// TIA Portal project "Paketband_6" (V20)

(* hardware
DEVICE "S7-1500/ET200MP-Station_1"  S7-1500 station
   slot 0: "Profilschiene_0"  Rack  6ES7 590-1***0-0AA0
   slot 1: "PLC_1"  CPU 1513-1 PN  6ES7 513-1AM03-0AB0  V4.0
      slot 3: "CPU-Display_1"  6ES7591-1AA00-0AA0
      slot 32768: "PROFINET-Schnittstelle_1"  X1
         slot 32769: "Port_1"  X1 P1
         slot 32770: "Port_2"  X1 P2
      slot 34817: "Virtual CP interface port_1"  Virtual CP interface port  Virtual CP interface port FW V4.0
   slot 2: "DI 16x24VDC BA_1"  DI 16x24VDC BA  6ES7 521-1BH10-0AA0  V1.1
   slot 3: "DQ 16x24VDC/0.5A ST_1"  DQ 16x24VDC/0.5A ST  6ES7 522-1BH00-0AB0  V2.0
   slot 4: "AI 8xU/I/R/RTD BA_1"  AI 8xU/I/R/RTD BA  6ES7 531-7QF00-0AB0  V1.0
   slot 5: "AQ 8xU/I HS_1"  AQ 8xU/I HS  6ES7 532-5HF00-0AB0  V2.2
   slot 6: "AQ 2xU/I ST_1"  AQ 2xU/I ST  6ES7 532-5NB00-0AB0  V1.0
*)

// ===== PLC "PLC_1"  CPU 1513-1 PN =====

VAR_GLOBAL   // PLC tag table "Standard-Variablentabelle"
   "PlcLabConnectIn01" AT %ID32760 : DWord;
   "PlcLabConnectIn02" AT %ID32764 : DWord;
   "PlcLabConnectOut01" AT %QD32760 : DWord;
   "PlcLabConnectOut02" AT %QD32764 : DWord;
   "Förderband_an" AT %M1.2 : Bool;
   "Förderband_aus" AT %M1.3 : Bool;
   "NotAus_aktiv" AT %M1.1 : Bool;
   "Anlage_ein" AT %M1.0 : Bool;
   "Paket_erkannt" AT %M1.4 : Bool;
   "Temp_1" AT %M0.0 : Bool;
   "Temp_2" AT %M0.1 : Bool;
   "Clock_Byte" AT %MB100 : Byte;
   "Clock_10Hz" AT %M100.0 : Bool;
   "Clock_5Hz" AT %M100.1 : Bool;
   "Clock_2.5Hz" AT %M100.2 : Bool;
   "Clock_2Hz" AT %M100.3 : Bool;
   "Clock_1.25Hz" AT %M100.4 : Bool;
   "Clock_1Hz" AT %M100.5 : Bool;
   "Clock_0.625Hz" AT %M100.6 : Bool;
   "Clock_0.5Hz" AT %M100.7 : Bool;
   "Förderband_starten" AT %M1.5 : Bool;
   "Paketzahl_erreicht" AT %M1.6 : Bool;
END_VAR

VAR_GLOBAL   // PLC tag table "Eingänge"
   "S1" AT %E0.4 : Bool;   // Start-Taster
   "S2" AT %E0.5 : Bool;   // Stopp-Taster
   "S4" AT %E0.0 : Bool;   // Not-Aus Schalter
   "S0" AT %E0.1 : Bool;   // Betriebsschalter auf ein
   "S3" AT %E0.6 : Bool;   // Rücksetz-Taster
   "S5" AT %E1.0 : Bool;   // Wiedereinschalten Taster
   "1b1" AT %E1.1 : Bool;   // Lichttaster (Mitte)
   "2b1" AT %E1.2 : Bool;   // Lichttaster (Ende)
   "S6" AT %E0.7 : Bool;   // Wartung quittieren Taster
END_VAR

VAR_GLOBAL   // PLC tag table "Ausgänge"
   "S1_Licht" AT %A0.4 : Bool;   // Lampe des Start-Tasters
   "S2_Licht" AT %A0.5 : Bool;   // Lampe des Stopp-Tasters
   "M1" AT %A0.0 : Bool;   // Förderband
   "S3_Licht" AT %A0.6 : Bool;   // Lampe des Rücksetz-Tasters
   "H1" AT %A0.1 : Bool;   // Meldeleuchte (Grün)
   "H2" AT %A0.2 : Bool;   // Meldeleuchte (Gelb)
   "H3" AT %A0.3 : Bool;   // Meldeleuchte (Rot)
   "Rundumleuchte" AT %A0.7 : Bool;
   "Zähler" AT %AW30 : Int;
   "H4" AT %A1.0 : Bool;   // Meldeleuchte (Blau)
END_VAR

// folder: System blocks/Program resources

DATA_BLOCK "DB_Timer_EV_3s"   // DB1
{ S7_Optimized_Access := 'TRUE' }
AUTHOR : Simatic
FAMILY : IEC
NAME : IEC_TMR
VERSION : 1.0
// stored: InstanceOfName IEC_TIMER
"IEC_TIMER"
BEGIN
END_DATA_BLOCK

DATA_BLOCK "DB_Timer_10d_Wartung"   // DB2
{ S7_Optimized_Access := 'TRUE' }
AUTHOR : Simatic
FAMILY : IEC
NAME : IEC_TMR
VERSION : 1.0
// stored: InstanceOfName IEC_TIMER
"IEC_TIMER"
BEGIN
END_DATA_BLOCK

DATA_BLOCK "DB_Timer_EV_2s"   // DB3
{ S7_Optimized_Access := 'TRUE' }
AUTHOR : Simatic
FAMILY : IEC
NAME : IEC_TMR
VERSION : 1.0
// stored: InstanceOfName IEC_TIMER
"IEC_TIMER"
BEGIN
END_DATA_BLOCK

DATA_BLOCK "DB_Counter_Pakete"   // DB4
{ S7_Optimized_Access := 'TRUE' }
AUTHOR : Simatic
FAMILY : IEC
NAME : CNTR
VERSION : 1.0
// stored: InstanceOfName IEC_COUNTER
"IEC_COUNTER"
BEGIN
END_DATA_BLOCK

// folder: (top level)

FUNCTION "Paketbandanlage" : Void   // FC1, FBD
{ S7_Optimized_Access := 'FALSE' }
VERSION : 0.1
   VAR_TEMP   // added for the SCL form of the ladder/FBD networks
      _w1 : Bool;
      _w2 : Bool;
   END_VAR
BEGIN

REGION Network 1: Paketbandsteuerung
   // Hinweis: Alle Schalter können nur benutzt werden, wenn die Anlage über den Betriebsschalter eingeschaltet wurde.
   // Über S2 (Stopp-Taster), 1b1 bzw. 2b1 (Lichttaster) wird das Paketband gestoppt. Der Stopp-Modus, wird durch start des Förderbandes deaktiviert.
   // Beide Modi (Start, Stopp) werden deaktiviert, sobald S4 (Not-Aus Schalter) aktiv ist.
   // Der Not-Aus-Modus kann nur über S3 (Rücksetz-Taster) deaktiviert werden.
   // Nach 10 Tagen Laufzeit des Förderbandes soll das Band kontrolliert werden, dazu soll die Rundumleuchte dann angehen. Mit S6 (Rücksetztaster) soll die Wartung quittiert werden.
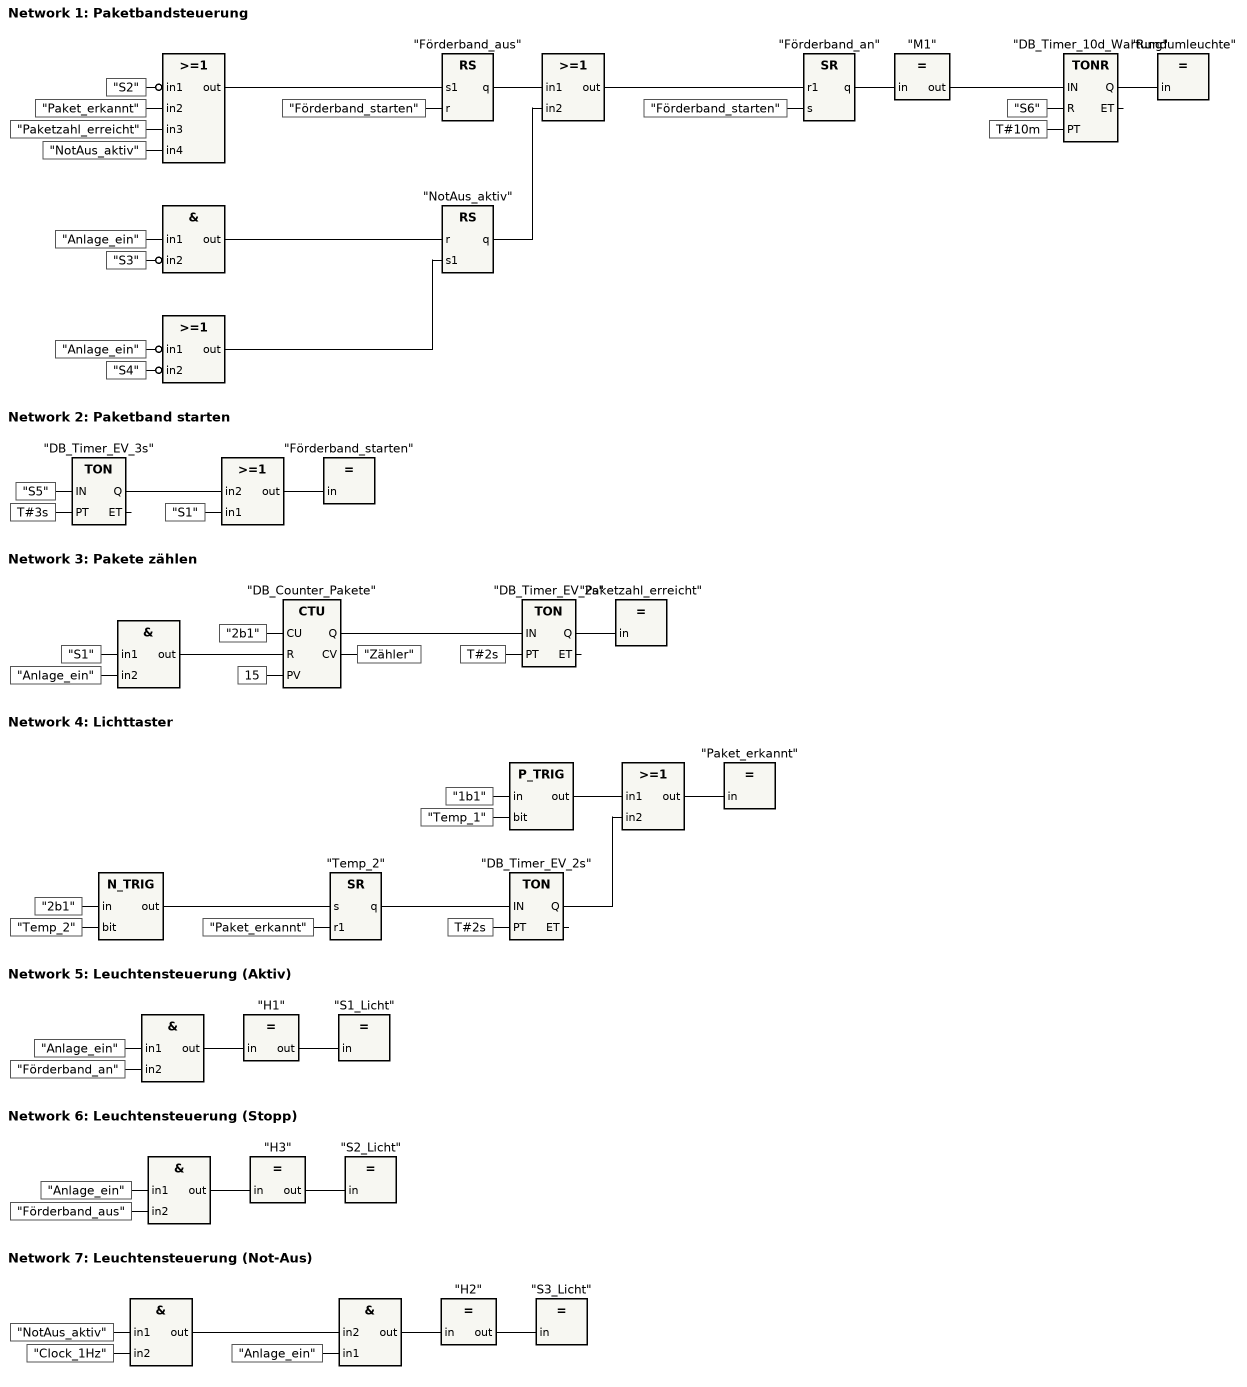
   IF "Förderband_starten" THEN
       "Förderband_aus" := FALSE;   // RS flip-flop
   END_IF;
   IF NOT "S2" OR "Paket_erkannt" OR "Paketzahl_erreicht" OR "NotAus_aktiv" THEN
       "Förderband_aus" := TRUE;
   END_IF;
   IF "Anlage_ein" AND NOT "S3" THEN
       "NotAus_aktiv" := FALSE;   // RS flip-flop
   END_IF;
   IF NOT "Anlage_ein" OR NOT "S4" THEN "NotAus_aktiv" := TRUE; END_IF;
   IF "Förderband_starten" THEN
       "Förderband_an" := TRUE;   // SR flip-flop
   END_IF;
   IF "Förderband_aus" OR "NotAus_aktiv" THEN "Förderband_an" := FALSE; END_IF;
   "M1" := "Förderband_an";
   "DB_Timer_10d_Wartung".TONR(IN := "Förderband_an", R := "S6", PT := T#10m);
   "Rundumleuchte" := "DB_Timer_10d_Wartung".Q;
END_REGION

REGION Network 2: Paketband starten
   // Das Paketband kann über S1 (Start-Taster) eingeschaltet werden bzw. durch S5 (Wiedereinschalten) und läuft dann dauerhaft. Der Schalter S5 (Wiedereinschalten) muss 3S gedrückt werden, bevor die Anlage wieder anlaufen darf. S1 (Starttaster) soll ganz normal funktionieren.
   "DB_Timer_EV_3s".TON(IN := "S5", PT := T#3s);
   "Förderband_starten" := "DB_Timer_EV_3s".Q OR "S1";
END_REGION

REGION Network 3: Pakete zählen
   // Nachdem 15 Pakete den hinteren Sensor durchlaufen haben, soll die Anlage automatisch abschalten. Über S1 (den Starttaster) soll der Zähler zurückgesetzt werden.
   "DB_Counter_Pakete".CTU(CU := "2b1", R := "S1" AND "Anlage_ein", PV := 15, CV => "Zähler");
   "DB_Timer_EV_2s".TON(IN := "DB_Counter_Pakete".Q, PT := T#2s);
   "Paketzahl_erreicht" := "DB_Timer_EV_2s".Q;
END_REGION

REGION Network 4: Lichttaster
   // Wenn 2b1 (der Lichttaster am Ende) oder 1b1 (Lichttaster in der Mitte) ein Paket erkennen, soll sofort bzw. verzögert das Band stehen bleiben.
   #_w1 := "1b1" AND NOT "Temp_1";   // rising edge
   "Temp_1" := "1b1";
   #_w2 := NOT "2b1" AND "Temp_2";   // falling edge
   "Temp_2" := "2b1";
   IF #_w2 THEN
       "Temp_2" := TRUE;   // SR flip-flop
   END_IF;
   IF "Paket_erkannt" THEN "Temp_2" := FALSE; END_IF;
   "DB_Timer_EV_2s".TON(IN := "Temp_2", PT := T#2s);
   "Paket_erkannt" := #_w1 OR "DB_Timer_EV_2s".Q;
END_REGION

REGION Network 5: Leuchtensteuerung (Aktiv)
   // Wenn die Anlage ein ist und gestartet wurde, dann soll die Meldeleuchte und die Leuchte des Start-Tasters leuchten.
   "H1" := "Anlage_ein" AND "Förderband_an";
   "S1_Licht" := "H1";
END_REGION

REGION Network 6: Leuchtensteuerung (Stopp)
   // Wenn die Anlage ein ist, aber gestoppt wurde, dann soll die Meldeleuchte und die Leuchte des Stopp-Tasters leuchten.
   "H3" := "Anlage_ein" AND "Förderband_aus";
   "S2_Licht" := "H3";
END_REGION

REGION Network 7: Leuchtensteuerung (Not-Aus)
   // Wenn die Anlage ein ist und sich im Not-Aus befindet, dann soll die Meldeleuchte und die Leuchte des Rücksetz-Tasters blinken.
   "H2" := "NotAus_aktiv" AND "Clock_1Hz" AND "Anlage_ein";
   "S3_Licht" := "H2";
END_REGION

REGION Network 8: Leuchtensteuerung (Mengenkontrolle)
   // Wenn die Anlage ein ist, dann soll die Meldeleuchte die produzierte Menge visualisieren. (<5 = aus, >5 = blinken, >10 = leuchten).
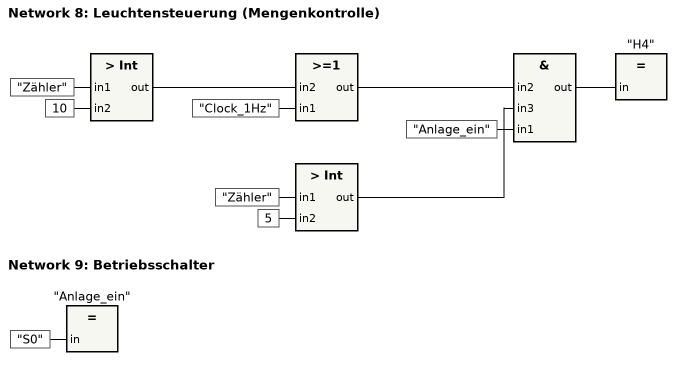
   "H4" := (("Zähler" > 10) OR "Clock_1Hz") AND ("Zähler" > 5) AND "Anlage_ein";
END_REGION

REGION Network 9: Betriebsschalter
   // Wenn der Betriebsschalter auf ein steht, sollen bestimmte Funktionsweisen möglich sein.
   "Anlage_ein" := "S0";
END_REGION
END_FUNCTION

ORGANIZATION_BLOCK "Main"   // OB1, FBD, ProgramCycle
TITLE = "Main Program Sweep (Cycle)"
{ S7_Optimized_Access := 'TRUE' }
VERSION : 0.1
   VAR_INPUT
      Initial_Call : Bool;   // Initial call of this OB
      Remanence : Bool;   // =True, if remanent data are available
   END_VAR
BEGIN

REGION Network 1
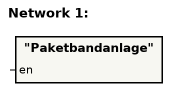
   "Paketbandanlage"();
END_REGION
END_ORGANIZATION_BLOCK